(* Logix 5000 project; controller PLC2_Project_1 Emulate 5570 rev 20.11; software revision 20.00 *)

TASK MainTask (continuous, watchdog 500 ms) : MainProgram

MODULES
   Local : Emulate 5570 (ICP 1, rev 20.11)
      Simulator_Card : vendor 1 type 0 code 15 (ICP 2, rev 1.1, Output RPI 50 ms)
END_MODULES

PROGRAM MainProgram   (* main routine MainRoutine *)
VAR
   Light_En : BOOL;
   Light_Start_Bit : BOOL;
   Light_Start_Delay : TIMER := (PRE := 1000);
   Light_Stop_Bit : BOOL;
   Light_Stop_Delay : TIMER := (PRE := 1000, ACC := 1039, EN := 1, DN := 1);
   ONS_Light_Start : BOOL;
   ONS_Light_Stop : BOOL := 1;
   ONS_Pump_Start : BOOL := 1;
   ONS_Pump_Stop : BOOL;
   PSI_H : BOOL;
   Pump_En : BOOL := 1;
   Pump_Off_Delay : TIMER := (PRE := 5000);
   Pump_Start_Bit : BOOL;
   Pump_Start_Delay : TIMER := (PRE := 5000, ACC := 5011, EN := 1, DN := 1);
   Pump_Stop_Bit : BOOL;
   Switch_110_PSI_Bit : BOOL;
   Switch_90_PSI_Bit : BOOL;
END_VAR

ROUTINE Controls   (* ladder *)
// Control program for the project
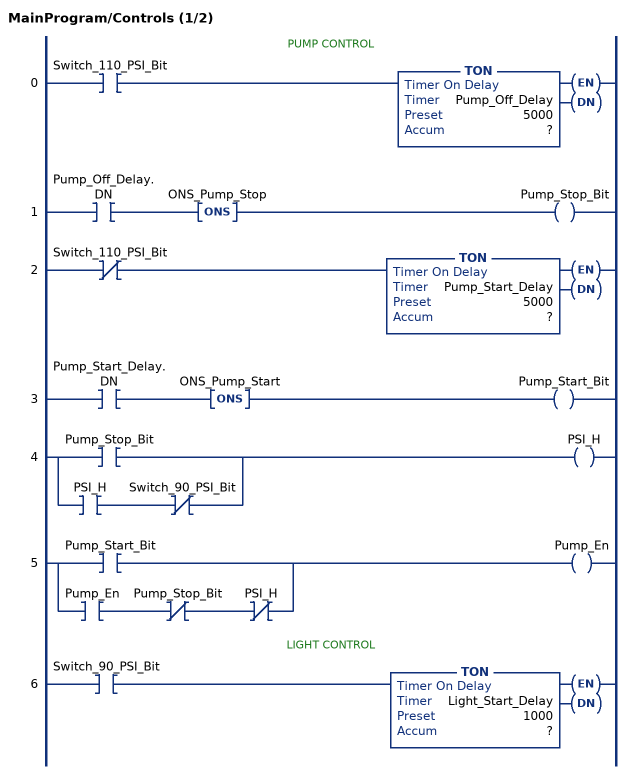
   // PUMP CONTROL
   0: XIC(Switch_110_PSI_Bit)TON(Pump_Off_Delay,?,?);
   1: XIC(Pump_Off_Delay.DN)ONS(ONS_Pump_Stop)OTE(Pump_Stop_Bit);
   2: XIO(Switch_110_PSI_Bit)TON(Pump_Start_Delay,?,?);
   3: XIC(Pump_Start_Delay.DN)ONS(ONS_Pump_Start)OTE(Pump_Start_Bit);
   4: [XIC(Pump_Stop_Bit) ,XIC(PSI_H) XIO(Switch_90_PSI_Bit) ]OTE(PSI_H);
   5: [XIC(Pump_Start_Bit) ,XIC(Pump_En) XIO(Pump_Stop_Bit) XIO(PSI_H) ]OTE(Pump_En);
   // LIGHT CONTROL
   6: XIC(Switch_90_PSI_Bit)TON(Light_Start_Delay,?,?);
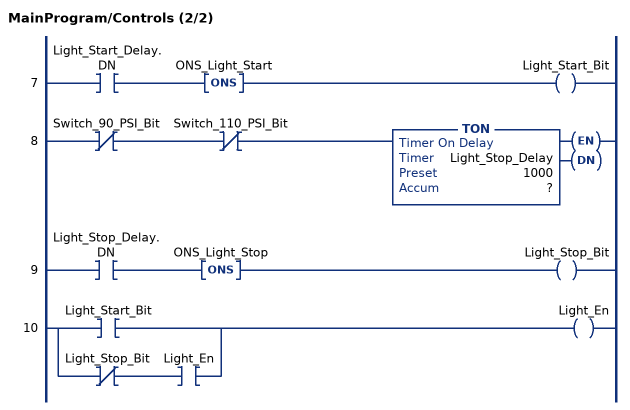
   7: XIC(Light_Start_Delay.DN)ONS(ONS_Light_Start)OTE(Light_Start_Bit);
   8: XIO(Switch_90_PSI_Bit)XIO(Switch_110_PSI_Bit)TON(Light_Stop_Delay,?,?);
   9: XIC(Light_Stop_Delay.DN)ONS(ONS_Light_Stop)OTE(Light_Stop_Bit);
   10: [XIC(Light_Start_Bit) ,XIO(Light_Stop_Bit) XIC(Light_En) ]OTE(Light_En);
END_ROUTINE

ROUTINE InputOutput   (* ladder *)
// All digital inputs & outputs
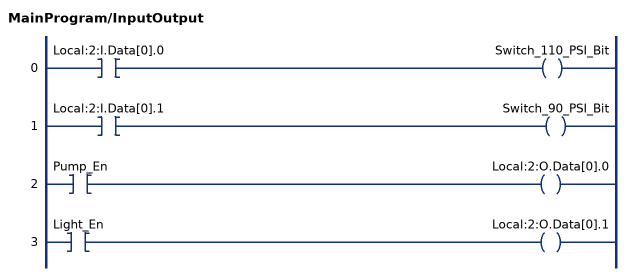
   0: XIC(Local:2:I.Data[0].0)OTE(Switch_110_PSI_Bit);
   1: XIC(Local:2:I.Data[0].1)OTE(Switch_90_PSI_Bit);
   2: XIC(Pump_En)OTE(Local:2:O.Data[0].0);
   3: XIC(Light_En)OTE(Local:2:O.Data[0].1);
END_ROUTINE

ROUTINE MainRoutine   (* ladder *)
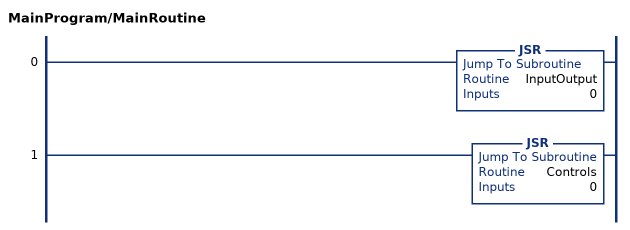
   0: JSR(InputOutput,0);
   1: JSR(Controls,0);
END_ROUTINE
END_PROGRAM
